(* IEC 61131-3 sources: programs/VI-54/VI-54_20171205/VI-54_20171205/Stations/Screen/LseClass170718/Class/RobotDimensions, 1 file *)

(* ---- RobotDimensions.st ---- *)
(*!
<Class
	Name               = "RobotDimensions"
	Revision           = "0.0"
	RealtimeTask       = "false"
	CyclicTask         = "false"
	BackgroundTask     = "false"
	Sigmatek           = "false"
	OSInterface        = "false"
	HighPriority       = "false"
	Automatic          = "false"
	UpdateMode         = "Prescan"
	SharedCommandTable = "true"
	Objectsize         = "(510,120)">
	<Channels>
		<Server Name="_________" Visualized="false" Initialize="false" WriteProtected="true" Retentive="false"/>
		<Server Name="__________" Visualized="false" Initialize="false" WriteProtected="true" Retentive="false"/>
		<Server Name="___________" Visualized="false" Initialize="false" WriteProtected="true" Retentive="false"/>
		<Server Name="Error_R_Pos" Visualized="false" Initialize="false" WriteProtected="true" Retentive="false"/>
		<Server Name="Error_X_Pos" Visualized="false" Initialize="false" WriteProtected="true" Retentive="false"/>
		<Server Name="Error_Y_Pos" Visualized="false" Initialize="false" WriteProtected="true" Retentive="false"/>
		<Server Name="Error_Z_Pos" Visualized="false" Initialize="false" WriteProtected="true" Retentive="false"/>
		<Server Name="Max_R" Visualized="true" Initialize="false" WriteProtected="false" Retentive="File"/>
		<Server Name="Max_X" Visualized="true" Initialize="false" WriteProtected="false" Retentive="File"/>
		<Server Name="Max_Y" Visualized="true" Initialize="false" WriteProtected="false" Retentive="File"/>
		<Server Name="Max_Z" Visualized="true" Initialize="false" WriteProtected="false" Retentive="File"/>
		<Server Name="Min_R" Visualized="true" Initialize="false" WriteProtected="false" Retentive="File"/>
		<Server Name="Min_X" Visualized="true" Initialize="false" WriteProtected="false" Retentive="File"/>
		<Server Name="Min_Y" Visualized="true" Initialize="false" WriteProtected="false" Retentive="File"/>
		<Server Name="Min_Z" Visualized="true" Initialize="false" WriteProtected="false" Retentive="File"/>
		<Client Name="ReadPositions" Required="true" Internal="false"/>
	</Channels>
</Class>
*)
RobotDimensions : CLASS
  //Servers:
	Max_X 	: SvrChCmd_DINT;
	Min_X 	: SvrCh_DINT;
	Error_X_Pos 	: SvrCh_DINT;
	__________ 	: SvrCh_DINT;
	Max_Y 	: SvrCh_DINT;
	Min_Y 	: SvrCh_DINT;
	Error_Y_Pos 	: SvrCh_DINT;
	___________ 	: SvrCh_DINT;
	Max_Z 	: SvrCh_DINT;
	Min_Z 	: SvrCh_DINT;
	Error_Z_Pos 	: SvrCh_DINT;
	_________ 	: SvrCh_DINT;
	Max_R 	: SvrCh_DINT;
	Min_R 	: SvrCh_DINT;
	Error_R_Pos 	: SvrCh_DINT;
  //Clients:
	ReadPositions 	: CltChCmd_ModelD4V2;
  //Variables:
		Xpositions 	: _LMCPROF_POS;
  //Functions:

	FUNCTION VIRTUAL GLOBAL Init;

	FUNCTION VIRTUAL GLOBAL CyWork
		VAR_INPUT
			EAX 	: UDINT;
		END_VAR
		VAR_OUTPUT
			state (EAX) 	: UDINT;
		END_VAR;

	FUNCTION GLOBAL ResetErrors;
  //Tables:
	FUNCTION @STD
		VAR_OUTPUT
			ret_code	: CONFSTATES;
		END_VAR;
	FUNCTION GLOBAL TAB @CT_;
END_CLASS;

#pragma usingLtd ModelD4V2

FUNCTION VIRTUAL GLOBAL RobotDimensions::Init

  // X dimensions
  if Min_X = 0 then
    Min_X := cX_SwMin;
  end_if;
  if Max_X = 0 then
    Max_X := cX_SwMax;
  end_if;

  // Y dimensions
  if Min_Y = 0 then
    Min_Y := cY_SwMin;
  end_if;
  if Max_Y = 0 then
    Max_Y := cY_SwMax;
  end_if;

  // Z dimensions
  if Min_Z = 0 then
    Min_Z := cZ_SwMin;
  end_if;
  if Max_Z = 0 then
    Max_Z := cZ_SwMax;
  end_if;

  // R dimensions
  if Min_R = 0 then
    Min_R := cR_SwMin;
  end_if;
  if Max_R = 0 then
    Max_R := cR_SwMax;
  end_if;

END_FUNCTION

FUNCTION VIRTUAL GLOBAL RobotDimensions::CyWork
	VAR_INPUT
		EAX 	: UDINT;
	END_VAR
	VAR_OUTPUT
		state (EAX) 	: UDINT;
	END_VAR

  ReadPositions.GetRobotPosition(Mode:=_LMCRobotBase::_POSITION_MODE::_ACTPOS_APPUNITS,
                                 IncludeTool:= False,
                                 CoordSystem:= 0,
                                 pPositions:= #Xpositions);

  // Check if X-position is in between the limits
  if Xpositions.Pos1 <= Max_X & Xpositions.Pos1 >= Min_X then
    Error_X_Pos := 0;
  else
  //  Error_X_Pos := 1;
  end_if;

  // Check if Y-position is in between the limits
  if Xpositions.Pos2 <= Max_Y & Xpositions.Pos2 >= Min_Y then
    Error_Y_Pos := 0;
  else
  //  Error_Y_Pos := 1;
  end_if;

  // Check if Z-position is in between the limits
  if Xpositions.Pos3 <= Max_Z & Xpositions.Pos3 >= Min_Z then
    Error_Z_Pos := 0;
  else
  //  Error_Z_Pos := 1;
  end_if;

  // Check if R-position is in between the limits
  if Xpositions.Pos4 <= Max_R & Xpositions.Pos4 >= Min_R then
    Error_R_Pos := 0;
  else
  //  Error_R_Pos := 1;
  end_if;

	state := READY;

END_FUNCTION

FUNCTION GLOBAL RobotDimensions::ResetErrors

  Error_X_Pos := 0;
  Error_Y_Pos := 0;
  Error_Z_Pos := 0;
  Error_R_Pos := 0;

END_FUNCTION
